// TwinCAT 3 PLC project BaseVistaSample
// ProgramVersion: 3.1.4020.1
// libraries:
//   Base_PLC,0.3.6.2,Vistaprint
//   Tc2_Standard,3.3.1.0,Beckhoff Automation GmbH
//   Tc2_System,3.4.13.0,Beckhoff Automation GmbH
//   Tc2_Utilities,3.3.14.0,Beckhoff Automation GmbH
//   Tc3_Interfaces,3.4.2.0,Beckhoff Automation GmbH
//   Tc3_MemMan,3.3.1.0,Beckhoff Automation GmbH
//   Tc3_Module,3.3.11.0,Beckhoff Automation GmbH
// project tree:
//   DUTs/ E_CtrlId.TcDUT, E_Test.TcDUT, E_TestWithNegatives.TcDUT, T_MetadataTest.TcDUT, T_PointerTest.TcDUT
//   GVLs/ Global.TcGVL, Io.TcGVL, Test.TcGVL
//   POUs/Controller/Lvl0/AGS %28Alarm Generator Simulator%29/ AGS_CmdState.TcGVL (not stored), FB_AGS.TcPOU (not stored), T_Ctrl_SIf_AGS.TcDUT (not stored), T_Ctrl_SIf_AGS_Cfg.TcDUT (not stored), T_Ctrl_SIf_AGS_Cur.TcDUT (not stored), T_Ctrl_SIf_AGS_In.TcDUT (not stored), T_Ctrl_SIf_AGS_Par.TcDUT (not stored)
//   POUs/Controller/Lvl0/CYL %28Exampel Cylinder use Base_Elements library for cylinders%29/ CYL_CmdState.TcGVL (not stored), E_ALM_CYL.TcDUT (not stored), E_Typ_CYL.TcDUT (not stored), FB_CYL.TcPOU (not stored), T_Ctrl_SIf_CYL.TcDUT (not stored), T_Ctrl_SIf_CYL_Cfg.TcDUT (not stored), T_Ctrl_SIf_CYL_Cur.TcDUT (not stored), T_Ctrl_SIf_CYL_Ilk.TcDUT (not stored), T_Ctrl_SIf_CYL_In.TcDUT (not stored), T_Ctrl_SIf_CYL_Out.TcDUT (not stored), T_Ctrl_SIf_CYL_Par.TcDUT (not stored)
//   POUs/Controller/Lvl2/MOD %28Modul%29/ E_ALM_MOD.TcDUT (not stored), E_Typ_MOD.TcDUT (not stored), FB_DtChnToLine_Test.TcPOU (not stored), FB_MOD.TcPOU (not stored), T_Ctrl_SIf_MOD.TcDUT (not stored), T_Ctrl_SIf_MOD_Cfg.TcDUT (not stored), T_Ctrl_SIf_MOD_Cur.TcDUT (not stored), T_Ctrl_SIf_MOD_DtChnToLine.TcDUT (not stored), T_Ctrl_SIf_MOD_DtChnToPLC.TcDUT (not stored), T_Ctrl_SIf_MOD_Ilk.TcDUT (not stored), T_Ctrl_SIf_MOD_Par.TcDUT (not stored)
//   POUs/Logger/StateLogger_FileClient/ FB_FileLc_StateLogger.TcPOU
//   POUs/Program/ FastPRG_1.TcPOU, MiddlePRG_1.TcPOU, SlowPRG_1.TcPOU
//   / Task_Fast.TcTTO, Task_Middle.TcTTO, Task_Slow.TcTTO
// real-time tasks:
//   TASK Task_Fast: cycle T#10ms, priority 5, ADS port 350
//   TASK Task_Slow: cycle T#80ms, priority 20, ADS port 351
//   TASK Task_Middle: cycle T#40ms, priority 10, ADS port 352

CONFIGURATION BaseVistaSample
    RESOURCE PLC ON TwinCAT3
        TASK Task_Fast(INTERVAL := T#10ms, PRIORITY := 5);
        TASK Task_Middle(INTERVAL := T#40ms, PRIORITY := 10);
        TASK Task_Slow(INTERVAL := T#80ms, PRIORITY := 20);
        PROGRAM FastPRG_1 WITH Task_Fast : FastPRG_1;
        PROGRAM MiddlePRG_1 WITH Task_Middle : MiddlePRG_1;
        PROGRAM SlowPRG_1 WITH Task_Slow : SlowPRG_1;
    END_RESOURCE
END_CONFIGURATION

// ---- DUTs/E_CtrlId.TcDUT
TYPE E_CtrlId :
(
	///not defined after startup...
	NONE,

	MOD_2,
	VER_2,
	HOR_2,
	AGS_1,
	AGS_2,

	E_CtrlIdMax
);
END_TYPE

// ---- DUTs/E_Test.TcDUT
// das ist ein test, kommentar ist direkt am ENUM typ, nicht an der instanz
TYPE E_Test :
(
	Empty := 0,
	STOP,
	LOAD,
	PICK,
	PRINT
);
END_TYPE

// ---- DUTs/E_TestWithNegatives.TcDUT
TYPE E_TestWithNegatives :
(
	Negative := -1,
	Zero := 0,
	One := 1,
	MAX_E_TestWithNegatives
);
END_TYPE

// ---- DUTs/T_MetadataTest.TcDUT
///
/// THIS STUCTURE IS USED FOR INTEGRATION TESTS
/// DO NOT CHANGE ANY VARIABLE OR COMMENT!
///

TYPE T_MetadataTest :
STRUCT
	/// a useful comment for the user (strSingleCommentTest)
	strSingleCommentTest: STRING;
	
	(*
		a useful comment for the user (strMultiCommentTest)
		with more details
	*)
	strMultiCommentTest: STRING;
	
	/// a useful comment for the user (strCommentMetadataTest) {hidden}{simulation}
	strCommentMetadataTest: STRING;
	
	(*
		a useful comment for the user (strCommentMetadataTestMixed_m)
		
		{unit:ms}
		defines the unit for UI. The unit in PLC might be different, in this case a conversion is necessary
		
		{range:0-999}
		limits the range in UI. User cannot enter values exceeding the range.
		
		{offset:5.8}
		shifts the value by an offset in UI
		
		{hidden}
		hides the Parameter/Configuration in UI except for the "saber" user who can see everything
		
		{readptr}
		tells the TagImporter to follow a pointer/reference and read out the de-referenced type. can be recursive. must be smart enough to detect cyclic pointers and break
	*)
	strCommentMetadataTestMixed_m: STRING;
	
	(*
		a useful comment for the user (eEnumTest)
		
		{enum 0=Empty;1=Stop;2=Load;3=Pick;4=Print}
		enum maps a useful text to the enumeration value. Useful for UI
	*)
	eEnumTest : E_Test;
	
	(*
		a useful comment for the user (eEnumWithNegativesTest)
		
		{enum
			-1=Negative;
			0=Zero;
			1=One}
	*)
	eEnumWithNegativesTest : E_TestWithNegatives;
END_STRUCT
END_TYPE

// ---- DUTs/T_PointerTest.TcDUT
TYPE T_PointerTest :
STRUCT
	bolPrintOk: BOOL;
	lreActTrayPos_mm : LREAL;
	eState: E_Test;	
END_STRUCT
END_TYPE

// ---- GVLs/Global.TcGVL
VAR_GLOBAL
	g_a_pCtrlInst: ARRAY[0..E_CtrlId.E_CtrlIdMax] OF POINTER TO fb_CtrlBase; // instance array of all controller instances
	g_a_pCtrlCIf: ARRAY[0..E_CtrlId.E_CtrlIdMax] OF POINTER TO T_Ctrl_CIf; // common interface array of all controllers (main use for PLC)
	g_p_fbAlm_Man: POINTER TO FB_Alm_Man; // common access variabel for UI

	g_uinStartProzess : UINT; // For StartUp order
  	// global base log
	g_fbBasLog: FB_BasLog; // only one central FB_BasLog instance/system allowed per PLC!!!
	// global file client
	g_fbFileLC: FB_FileLc; // only one central FB_FileLc instance allowed per PLC!!!
	g_bolLogEnableState : BOOL := TRUE; // EnableState log
	
END_VAR

VAR_GLOBAL CONSTANT
	c_uinCntTaskClass : UINT := 3;	// Count of Task Classes
END_VAR

// ---- GVLs/Io.TcGVL
VAR_GLOBAL
	///input fb instance Cyl_AB position retract normally open
	In_bolHOR_2_Retracted_NO AT %I* : BOOL;
	///input fb instance Cyl_AB position extend normally closed
	In_bolHOR_2_Extended_NC AT %I*: BOOL;
	///output fb instance Cyl_AB valve retract
	Out_bolHOR_2_Retract AT %Q* : BOOL;
	///output fb instance Cyl_AB valve extend
	Out_bolHOR_2_Extend AT %Q* : BOOL;
END_VAR

// ---- GVLs/Test.TcGVL
// This file does not demonstrate the PLC BaseVista concept. It's used for PlcCommunication testing.
VAR_GLOBAL
	strDefaultString	: STRING;
	strLongString		: STRING(160);
	strShortString		: STRING(5);
	
	bolTest		: BOOL;
END_VAR

// ---- POUs/Program/FastPRG_1.TcPOU
PROGRAM FastPRG_1
VAR

END_VAR

(*__________________________________________________________________________________________________
¦	
¦	Vistaprint Schweiz GmbH
¦	CH - 8401 Winterthur
¦
¦	www.vistaprint.ch - info@vistaprint.ch
¦___________________________________________________________________________________________________

Function desription:
call of all controller (FUB) for the fast task class.


History:
Version		Date			Author		Comment
---------------------------------------------------------------------------------------------------
0.00.1		25.05.2013		AVME/KVO	Start history


___________________________________________________________________________________________________*)


// -----------------------------------------------------------------------------------------------
// Initialize the PLC Parameter and check the PLC health
// -----------------------------------------------------------------------------------------------
IF (g_uinStartProzess=0) THEN
	g_uinStartProzess:=1; // For StartUp order

END_IF
// -----------------------------------------------------------------------------------------------


// -----------------------------------------------------------------------------------------------
// The host system is downloading all parameter at startup. 
// bolPlcStartupDone will be set to true after the Host is done with the initialization
// -----------------------------------------------------------------------------------------------
IF (g_uinStartProzess=c_uinCntTaskClass) THEN
	g_uinStartProzess := 11; // For StartUp order
END_IF
// -----------------------------------------------------------------------------------------------


// -----------------------------------------------------------------------------------------------
// Start PLC code initialization
// -----------------------------------------------------------------------------------------------
IF (g_uinStartProzess=(10+c_uinCntTaskClass)) THEN
	
	// init	
	g_uinStartProzess := 21; // For StartUp order
END_IF
// -----------------------------------------------------------------------------------------------


// -----------------------------------------------------------------------------------------------
// Normal Run mode after1 all the initialization is done
// -----------------------------------------------------------------------------------------------
IF (g_uinStartProzess>=(20+c_uinCntTaskClass)) THEN
	;
END_IF
// -----------------------------------------------------------------------------------------------

END_PROGRAM

// ---- POUs/Program/MiddlePRG_1.TcPOU
PROGRAM MiddlePRG_1
VAR
	uinTaskNbr : UINT := 2; // MiddleTask is Task Nr. 2
	fbMOD_2: FB_MOD;
	fbVER_2: FB_CYL;
	fbHOR_2: FB_CYL;
	
	stTest : T_PointerTest;
	fbAGS_1: FB_AGS;
	fbAGS_2: FB_AGS;
	
	fbDLL_1: BASE_PLC.FB_DLL(In_bDoDataWipe:=FALSE);
	
END_VAR

(*__________________________________________________________________________________________________
¦	
¦	Vistaprint Schweiz GmbH
¦	CH - 8401 Winterthur
¦
¦	www.vistaprint.ch - info@vistaprint.ch
¦___________________________________________________________________________________________________

Function desription:
call of all controller (FUB) for the middel task class inclusiv alarm handler.


History:
Version		Date			Author		Comment
---------------------------------------------------------------------------------------------------
0.00.1		02.05.2013		AVME/KVO	Start history


___________________________________________________________________________________________________*)

// -----------------------------------------------------------------------------------------------
// Initialize the PLC Parameter and check the PLC health
// -----------------------------------------------------------------------------------------------
IF (g_uinStartProzess=(uinTaskNbr-1)) THEN
	// init
	//Driver
	
	//Lvl0
	fbHOR_2.iniAllCtrlArrays(ADR(g_a_pCtrlInst),ADR(g_a_pCtrlCIf),E_CtrlId.HOR_2); // init and entry fb_instance and adr of ctrl interface struct in global pointer arrays
	fbVER_2.iniAllCtrlArrays(ADR(g_a_pCtrlInst),ADR(g_a_pCtrlCIf),E_CtrlId.VER_2); // init and entry fb_instance and adr of ctrl interface struct in global pointer arrays

	fbAGS_1.iniAllCtrlArrays(ADR(g_a_pCtrlInst),ADR(g_a_pCtrlCIf),E_CtrlId.AGS_1);
	fbAGS_1.ptrPointerTest := ADR(stTest);
	fbAGS_1.ptrCircularPointerTest := ADR(fbAGS_2);
	stTest.bolPrintOk := TRUE;
	stTest.lreActTrayPos_mm := 10;
	
	fbAGS_2.iniAllCtrlArrays(ADR(g_a_pCtrlInst),ADR(g_a_pCtrlCIf),E_CtrlId.AGS_2);
	fbAGS_2.ptrCircularPointerTest := ADR(fbAGS_1);
	
	//Lvl2
	fbMOD_2.iniAllCtrlArrays(ADR(g_a_pCtrlInst),ADR(g_a_pCtrlCIf),E_CtrlId.MOD_2);  // init and entry fb_instance and adr of ctrl interface struct in global pointer arrays
	// add childs
	fbMOD_2.In_p_fbHOR := g_a_pCtrlInst[E_CtrlId.HOR_2];
	fbMOD_2.In_p_fbVER := g_a_pCtrlInst[E_CtrlId.VER_2];
	
	g_uinStartProzess := g_uinStartProzess + 1; // For StartUp order
END_IF
// -----------------------------------------------------------------------------------------------


// -----------------------------------------------------------------------------------------------
// The host system is downloading all parameter at startup. 
// bolPlcStartupDone will be set to true after the Host is done with the initialization
// -----------------------------------------------------------------------------------------------
IF (g_uinStartProzess=(uinTaskNbr-1)+10) THEN
	g_uinStartProzess := g_uinStartProzess + 1; // For StartUp order
END_IF
// -----------------------------------------------------------------------------------------------


// -----------------------------------------------------------------------------------------------
// Start PLC code initialization
// -----------------------------------------------------------------------------------------------
IF (g_uinStartProzess=(uinTaskNbr-1)+20) THEN
	
	// init
	fbMOD_2.CtrlCIf^.Job.intACmd := cCMD_RUN;
	
	g_uinStartProzess := g_uinStartProzess + 1; // For StartUp order
END_IF
// -----------------------------------------------------------------------------------------------



// -----------------------------------------------------------------------------------------------
// Normal Run mode after all the initialization is done
// -----------------------------------------------------------------------------------------------
IF (g_uinStartProzess>=(20+c_uinCntTaskClass)) THEN
	
	//****************************************************************************************************
	// cyclic controller calls
	//****************************************************************************************************

	// Modul example
	// ----------------------------------------------------------------------------------------------------------------------------
	// modul controller MOD_2 with childs
	fbMOD_2();
	fbVER_2();
	
	fbHOR_2.In_bolRetracted := In_bolHOR_2_Retracted_NO;
	fbHOR_2.In_bolExtended := (NOT In_bolHOR_2_Extended_NC);
	fbHOR_2();
	Out_bolHOR_2_Retract := fbHOR_2.Out_bolRetract;
	Out_bolHOR_2_Extend := fbHOR_2.Out_bolExtend;
	
	fbAGS_1();

END_IF
// -----------------------------------------------------------------------------------------------

END_PROGRAM

// ---- POUs/Program/SlowPRG_1.TcPOU
PROGRAM SlowPRG_1
VAR
	uinTaskNbr : UINT := 3; // SlowTask is Task Nr 3
	jj:INT;
	bolCtrlRst: BOOL;
	bolInitAllCtrlDone : BOOL := FALSE;
	
	fbAlm_Man: FB_Alm_Man; // alarm manager
	fbFileLc_StateLogger : FB_FileLc_StateLogger; // file client for state logger
	
	/// Switches all controllers in loading station to simulation with pos. edge
	bolSimulateAll: BOOL;
	bolSimulationActive: BOOL;
	
	// for tests
	intCmd : INT;
	stFileTime : T_FILETIME;
	stTimeStruct : TIMESTRUCT;
	fbQueueTest_Receiver : FB_QueueTest_Receiver;
	fbBasLogTest_Client: FB_BasLogTest_Client;
	fbBasLogTest_Sender : FB_BasLogTest_Sender;
	fbFileLcTest:	FB_FileLcTest;
	fbTimeStamp: FB_TimeStamp;
END_VAR

(*__________________________________________________________________________________________________
¦	
¦	Vistaprint Schweiz GmbH
¦	CH - 8401 Winterthur
¦
¦	www.vistaprint.ch - info@vistaprint.ch
¦___________________________________________________________________________________________________

Function desription:
call of all controller (FUB) for the slow task class.


History:
Version		Date			Author		Comment
---------------------------------------------------------------------------------------------------
0.00.1		24.05.2013		AVME/KVO	Start history
0.00.2		07.11.2013		AVME/KVO	Add local variabel fbAlm_Man, Add set all initialized controller FB the property of the alarm manager adress 
0.00.3		08.11.2013		AVME/KVO	global g_p_fbAlm_Man adress assigned
0.00.4		17.02.2014		AVME/KVO	startup check init FB_Alarm IsInitDone
0.00.5		15.10.2014		AVME/KVO	Add StateLogger file client call and add setAllCtrlBasLogFB
										Add Simulate all - standard new simulation = false!
___________________________________________________________________________________________________*)


// -----------------------------------------------------------------------------------------------
// Initialize the PLC Parameter and check the PLC health
// -----------------------------------------------------------------------------------------------
IF (g_uinStartProzess=(uinTaskNbr-1)) THEN
	//*************** only call onetime!!!! after init all controllers before!!!*******************************
	IF (bolInitAllCtrlDone=FALSE) THEN
		// set all initialized controller FB the property of the alarm manager adress 
		// set all initialized controller FB the property of the base logger system adress 
		// call all CtrlInit()
		Base_PLC.initAllCtrl(pCtrlInst := ADR(g_a_pCtrlInst[0]), pBasLogFB := ADR(g_fbBasLog), pAlarmCtrl := ADR(fbAlm_Man), uinCtrlInstLength := INT_TO_UINT(E_CtrlId.E_CtrlIdMax));
		bolInitAllCtrlDone := TRUE;
	END_IF
	
	g_p_fbAlm_Man := ADR(fbAlm_Man);
	
	// for sample - simulation activation automatic
	bolSimulateAll := TRUE;
	
	//****************************************************************************************************
	// Log system - init file client's - takes more than one cycle!
	//****************************************************************************************************
	// state logger file client: init -> readout config file, allocate memory -> cyclic read out state logs and write to csv file
	fbFileLc_StateLogger(In_p_fbBasLog:=ADR(g_fbBasLog),In_p_fbFileLC:=ADR(g_fbFileLc));
	
	IF (fbFileLc_StateLogger.Out_bolInitDone=TRUE) OR  (g_bolLogEnableState = FALSE)  THEN
		// test file client: init -> readout config file, allocate memory -> cyclic read out state logs and write to csv file
		fbFileLcTest.In_strPath := 'C:\Vistaprint\Log\';
		fbFileLcTest.In_strCfgFileName := 'StateLogTest.cfg';
		fbFileLcTest.In_p_fbBasLog := ADR(g_fbBasLog);
		fbFileLcTest.In_p_fbFileLC := ADR(g_fbFileLC);
		fbFileLcTest();

		IF (fbFileLcTest.Out_bolInitDone=TRUE) THEN
			g_uinStartProzess := g_uinStartProzess + 1; // For StartUp order
		END_IF
	END_IF
END_IF
// -----------------------------------------------------------------------------------------------


// -----------------------------------------------------------------------------------------------
// The host system is downloading all parameter at startup. 
// bolPlcStartupDone will be set to true after the Host is done with the initialization
// -----------------------------------------------------------------------------------------------
IF (g_uinStartProzess=(uinTaskNbr-1)+10) THEN
	g_uinStartProzess := g_uinStartProzess + 1; // For StartUp order
END_IF
// -----------------------------------------------------------------------------------------------


// -----------------------------------------------------------------------------------------------
// Start PLC code initialization
// -----------------------------------------------------------------------------------------------
IF (g_uinStartProzess=(uinTaskNbr-1)+20) THEN
	// init call alarm FB until init is done
	fbAlm_Man(bolCtrlRst:= bolCtrlRst);
	
	// init	
	IF (fbAlm_Man.IsInitDone = TRUE) THEN
		g_uinStartProzess := g_uinStartProzess + 1; // For StartUp order
	END_IF
END_IF
// -----------------------------------------------------------------------------------------------

// -----------------------------------------------------------------------------------------------
// Normal Run mode after all the initialization is done
// -----------------------------------------------------------------------------------------------
IF (g_uinStartProzess>=(20+c_uinCntTaskClass)) THEN
	//****************************************************************************************************
	// SIMULATE all controller
	//****************************************************************************************************
	IF (bolSimulateAll = TRUE) AND (bolSimulationActive = FALSE) THEN
		// Enable simulation for all controller	
		FOR jj:=0 TO E_CtrlId.E_CtrlIdMax BY 1 DO
			IF (g_a_pCtrlCIf[jj]<>0) THEN // check if entry exist
				g_a_pCtrlCIf[jj]^.SwCfg.bolSimulation := TRUE;
			END_IF
		END_FOR	
		bolSimulationActive:= TRUE;
		// Trigger an alarm reset
		bolCtrlRst:= TRUE;
	END_IF
		
	IF (bolSimulateAll = FALSE) AND (bolSimulationActive = TRUE) THEN
		// Disable simulation for all controller	
		FOR jj:=0 TO E_CtrlId.E_CtrlIdMax BY 1 DO
			IF (g_a_pCtrlCIf[jj]<>0) THEN // check if entry exist
				g_a_pCtrlCIf[jj]^.SwCfg.bolSimulation := FALSE;
			END_IF
		END_FOR	
		bolSimulationActive:= FALSE;		
	END_IF

	//****************************************************************************************************
	// call alarm message handler
	//****************************************************************************************************
	fbAlm_Man(bolCtrlRst:= bolCtrlRst);
	IF (bolCtrlRst) THEN
		FOR jj:=0 TO E_CtrlId.E_CtrlIdMax BY 1 DO
			IF (g_a_pCtrlCIf[jj]<>0) THEN // check if entry exist
				g_a_pCtrlCIf[jj]^.Job.bolAlmReset := TRUE;
			END_IF
		END_FOR
		bolCtrlRst := FALSE;
	END_IF
	
	//****************************************************************************************************
	// file client call for state logger
	//****************************************************************************************************
	fbFileLc_StateLogger();
	IF (fbFileLc_StateLogger.Out_udiStatus<>0) THEN // state log file client error
		;
		//fbAlm_Man.setAlarm(p_fbMAIN^.CtrlCIf^.Info.intCtrlId,E_ALM_MAIN.ViperLogFileClient,UDINT_TO_DINT(fbFileClient_ViperLog.Out_udiStatus),ADR(pTmpSIf_MAIN^.Alm),E_AlmState.RST,p_fbMAIN^.CtrlCIf^.Job.eMe_ActivAlmClass);
	END_IF
	// ***********************************************************************************************
	// Test file client
	fbFileLcTest();
	IF (fbFileLcTest.Out_udiStatus<>0) THEN // state log file client error
		;
		//fbAlm_Man.setAlarm(p_fbMAIN^.CtrlCIf^.Info.intCtrlId,E_ALM_MAIN.ViperLogFileClient,UDINT_TO_DINT(fbFileClient_ViperLog.Out_udiStatus),ADR(pTmpSIf_MAIN^.Alm),E_AlmState.RST,p_fbMAIN^.CtrlCIf^.Job.eMe_ActivAlmClass);
	END_IF
END_IF
// -----------------------------------------------------------------------------------------------


// ***********************************************************************************************
// only for sw-tests
// ***********************************************************************************************
// Test Base log system
fbBasLogTest_Sender(In_p_fbBasLog:= ADR(g_fbBasLog));
fbBasLogTest_Client(In_p_fbBasLog:= ADR(g_fbBasLog));

END_PROGRAM

// ---- POUs/Logger/StateLogger_FileClient/FB_FileLc_StateLogger.TcPOU

FUNCTION_BLOCK FB_FileLc_StateLogger
VAR_INPUT
	In_p_fbBasLog: POINTER TO FB_BasLog; // only one central FB_BasLog instance allowed per PLC!!!
	In_p_fbFileLC: POINTER TO FB_FileLc; // only one central FB_FileLc instance allowed per PLC!!!
END_VAR
VAR_OUTPUT
	Out_bolInitDone : BOOL;
	Out_udiStatus : UDINT;
END_VAR
VAR
	uinActFLcClientIdx : UINT; // file client index for init
	bolInit : BOOL := FALSE; // FALSE: autostart with init
	bolGetFirstHandle : BOOL;
	bolDone : BOOL;
	udiInitStatus : UDINT;
	udiStatus : UDINT;
	pHandle : POINTER TO T_FileLc_SysInfo;
	// for test send
	pHandleBaseLog : POINTER TO T_Bl_LibHandleRow;
	uinGetHandleBaseLogStatus : UINT;
	intDoWrite : INT;
	dinPar1 : DINT;
	strText1 : STRING(BasLog.cMAX_CHAR_TEXT1):='Statelogger test - Controller 1';
	strText2 : STRING(BasLog.cMAX_CHAR_TEXT2):='Statelogger test - sub info';
	uinWriteStatus : UINT;
END_VAR

(*__________________________________________________________________________________________________
¦	
¦	Vistaprint Schweiz GmbH
¦	CH - 8401 Winterthur
¦
¦	www.vistaprint.ch - info@vistaprint.ch
¦___________________________________________________________________________________________________

Function desription:
Function block capsule the state logger file client call in the application.

History:
Version		Date			Author		Comment
---------------------------------------------------------------------------------------------------
0.00.1		14.10.2014		AVME/KVO	Start history
___________________________________________________________________________________________________*)

IF (In_p_fbFileLC<>TC3_MEMMAN.NULL) AND (g_bolLogEnableState=TRUE) THEN // check if pointer valid
	
	// system init onetime after start up
	IF (Out_bolInitDone=FALSE) THEN
		In_p_fbFileLC^.M_Init(In_bolExecute := TRUE,In_p_uinFLcIdx := ADR(uinActFLcClientIdx),In_strCfgFileName:='StateLogCsv.cfg',In_strPath:='C:\Vistaprint\Log\',In_p_fbBasLog := In_p_fbBasLog,Out_pHandle=>pHandle,Out_udiStatus=>udiInitStatus,Out_bolDone=>bolDone);
		IF (bolDone OR (udiInitStatus<>0)) THEN
			// negative edge -> reinit possibel and release init next file client!!!
			In_p_fbFileLC^.M_Init(In_bolExecute := FALSE,In_p_uinFLcIdx := ADR(uinActFLcClientIdx),In_strCfgFileName:='StateLogCsv.cfg',In_strPath:='C:\Vistaprint\Log\',In_p_fbBasLog := In_p_fbBasLog);
			Out_bolInitDone := TRUE;
		END_IF
	ELSE
		IF ((pHandle<>TC3_MEMMAN.NULL) AND (udiInitStatus=0)) THEN	// valid pointer => init ok
			// cyclic call of file client - alarm generation in application if status not ok???
			udiStatus := In_p_fbFileLC^.M_Cyclic(In_pHandle:=pHandle);
			
			// *******************************************************************************************************************************************
			// only for sending test logs!!!
			// get write handle for tests
			IF (bolGetFirstHandle=FALSE) THEN
				uinGetHandleBaseLogStatus := In_p_fbBasLog^.M_GetHandle(Out_pHandle=>pHandleBaseLog);// fbBasLog global defined base log system fub (only once per system)
				bolGetFirstHandle := TRUE;
			END_IF
			
			// write test state log entries
			IF (pHandleBaseLog<>TC3_MEMMAN.NULL) AND (intDoWrite>0) THEN
				intDoWrite := intDoWrite - 1;
				dinPar1 := dinPar1 + 1;
				uinWriteStatus := In_p_fbBasLog^.M_Log(In_pHandle:=pHandleBaseLog,In_udiLogType:=BasLog.cLOGTYPE_STATELOG,In_intCtrlID:=11,In_strText1:=strText1,In_strText2:=strText2,In_dinPar1:=dinPar1,In_dinPar2:=0,In_dinPar3:=0,In_dinPar4:=0) ;
			END_IF
			// *******************************************************************************************************************************************
		END_IF;		
	END_IF

	// out for failures
	IF (udiInitStatus<>0)THEN
		Out_udiStatus := udiInitStatus;
	ELSE
		Out_udiStatus := udiStatus;
	END_IF
END_IF

END_FUNCTION_BLOCK
